{attribute 'qualified_only'}
{attribute 'strict'}
{attribute 'to_string'}
TYPE eGeneralState :
(
	Idle 		:= 0,
	Stopped 	:= 1,
	Aborted 	:= 2
);
END_TYPE

(* stored: Version 1.1.0.1
   DUT eGeneralState: Id {ed1ae5ce-6664-4b38-b3bc-3cb46a1a1274} *)
